TYPE ST_Powermodule_CalibData :
STRUCT
	Pset: ARRAY[0..4] OF REAL;
	Qset: ARRAY[0..4] OF REAL;
	Pmeas: ARRAY[0..4] OF ARRAY[0..4] OF REAL;
	Qmeas: ARRAY[0..4] OF ARRAY[0..4] OF REAL;
END_STRUCT
END_TYPE

(* stored: Version 1.1.0.1, ProductVersion 3.1.4026.18
   DUT ST_Powermodule_CalibData: Id {ae5fbc2e-b17f-4b3c-b7f5-ebd16fc257ab} *)
